// TwinCAT 3 PLC project Untitled1
// ProgramVersion: 3.1.4023.0
// libraries:
//   Tc2_MC2, * (Beckhoff Automation GmbH)
//   Tc2_Standard, * (Beckhoff Automation GmbH)
//   Tc2_System, * (Beckhoff Automation GmbH)
//   Tc3_Module, * (Beckhoff Automation GmbH)
// project tree:
//   DUTs/ AirPiston.TcPOU, ClearLinkEIP.TcPOU (not stored), Homing.TcDUT (not stored), PneumaticInsertion.TcPOU, SuctionPad.TcDUT (not stored)
//   / PlcTask.TcTTO
//   POUs/ MAIN.TcPOU, PistonOnly.TcPOU, WithinTolerance.TcPOU (not stored)
// real-time tasks:
//   TASK PlcTask: cycle T#10ms, priority 20, ADS port 350

CONFIGURATION Untitled1
    RESOURCE PLC ON TwinCAT3
        TASK PlcTask(INTERVAL := T#10ms, PRIORITY := 20);
        PROGRAM MAIN WITH PlcTask : MAIN;
    END_RESOURCE
END_CONFIGURATION

// ---- POUs/MAIN.TcPOU
PROGRAM MAIN
VAR
	insertion : PneumaticInsertion;
	
	enable : BOOL;
	up : BOOL;
	down : BOOL;
	
	in : BOOL;
	out : BOOL;
	
	suction : ARRAY[1..4] OF SuctionPad;
	enableAllSuction : BOOL;
	i : INT;
END_VAR

PistonOnly(smc := insertion.screw);

(*
insertion(
	enable:= enable, 
	slider=> , 
	screw=> , 
	contact=> , 
	home=> , 
	ready=> , 
	busy=> , 
	error=> , 
	homeSet=> );

IF NOT insertion.screw.homeSet THEN
	insertion.homingSequence();
	RETURN;
END_IF

insertion.stop();
	
IF in THEN
	insertion.press();
	out := FALSE;
END_IF

IF out THEN
	insertion.release();
	in := FALSE;
END_IF

IF up THEN
	insertion.slideContinuous(direction:= MC_Positive_Direction);
	down := FALSE;
END_IF

IF down THEN
	insertion.slideContinuous(direction:= MC_Negative_Direction);
	up := FALSE;
END_IF

IF enableAllSuction THEN
	FOR i:=1 TO 4 BY 1 DO
		suction[i].enable := TRUE;
	END_FOR
END_IF
*)

END_PROGRAM

// ---- DUTs/PneumaticInsertion.TcPOU
FUNCTION_BLOCK PneumaticInsertion// EXTENDS Insertion
VAR_INPUT
	enable : BOOL;
END_VAR
VAR_OUTPUT
	slider : ClearLinkEIP;
	screw : AirPiston;
	
	contact : BOOL;
	
	home : BOOL;
	ready : BOOL;
	busy : BOOL;
	error : BOOL;
	
	homeSet : BOOL;
END_VAR

slider(
	bEnable:= enable, 
	home=> , 
	outerLimit=> , 
	innerLimit=> , 
	contact=> contact, 
	homeSet=> );
	
screw(
	bEnable:= enable,
	valveExtend=> , 
	valveRetract=> , 
	contact=> , 
	home=> , 
	innerLimit=> , 
	ready=> , 
	busy=> , 
	error=> , 
	homeSet=> );
	
home := screw.home AND slider.home;
busy := slider.busy OR screw.busy;
error := slider.error OR screw.error;

homeSet := slider.homeSet AND screw.homeSet;

METHOD homingSequence : BOOL
IF NOT screw.homeSet THEN
	screw.homingSequence();
END_IF

homingSequence := slider.homeSet (*AND screw.homeSet*);
END_METHOD

METHOD press : BOOL
VAR_INPUT
	//direction : BOOL; //direction (F = inwards, T = outwards)
	//distance : DINT;
END_VAR
press := screw.extend();
END_METHOD

METHOD release : BOOL
VAR_INPUT
END_VAR
release := screw.retract();
END_METHOD

METHOD slideAbsolute : BOOL
VAR_INPUT
	targetPos : REAL;
END_VAR
slideAbsolute := slider.moveAbsolute(newTarget:= targetPos);
END_METHOD

METHOD slideContinuous : BOOL
VAR_INPUT
	direction : MC_Direction;
END_VAR
slideContinuous := slider.moveContinuous(direction := direction);
END_METHOD

METHOD stop : BOOL
VAR_INPUT
END_VAR
slider.stop();
screw.stop();
END_METHOD

END_FUNCTION_BLOCK

// ---- DUTs/AirPiston.TcPOU
FUNCTION_BLOCK AirPiston
VAR_INPUT CONSTANT
	bEnable : BOOL;
END_VAR
VAR_OUTPUT
	valveExtend AT %Q* : BOOL;
	valveRetract AT %Q* : BOOL;
	
	contact AT %I* : BOOL;
	
	home AT %I* : BOOL;
	innerLimit AT %I* : BOOL;
	
	ready : BOOL;
	busy : BOOL;
	error : BOOL;
	homeSet : BOOL;
END_VAR
VAR
	brakeMode : (PULSE, VARIABLE) := PULSE;
	brakePulse : TP;
	
	step : Homing;
	mode : (HOLD, IN, OUT, REVERSAL);
END_VAR
VAR_STAT CONSTANT
	brakeTime : TIME := T#500MS;
END_VAR

IF NOT bEnable THEN
	stop();
	RETURN;
END_IF

brakePulse(IN:= , PT:= brakeTime, Q=> , ET=> ); //reversal to act as brake
brakePulse.IN := brakePulse.IN AND brakePulse.Q; //automatically turn off pulse

IF home AND valveRetract THEN
	mode := HOLD;
	
ELSIF (innerLimit OR contact) AND valveExtend THEN
	
	IF brakeMode = PULSE THEN
		brakePulse.IN := TRUE; //start reversal to sensor inner limit
		mode := HOLD;
		
	ELSIF brakeMode = VARIABLE THEN
		mode := REVERSAL;
		//RETURN;
		
	END_IF
	
END_IF

CASE mode OF
	HOLD:
		valveExtend := FALSE;
		valveRetract := FALSE;
		
	IN:
		valveExtend := TRUE;
		valveRetract := FALSE;
		
	OUT:
		valveExtend := FALSE;
		valveRetract := TRUE;
		
	REVERSAL:		
		valveExtend := FALSE;
		valveRetract := TRUE;
		
		IF innerLimit THEN
			mode := HOLD;
		END_IF
		
END_CASE

valveRetract := valveRetract OR brakePulse.Q; //from mode or brake

METHOD extend : BOOL
VAR_INPUT
END_VAR
mode := IN;
END_METHOD

METHOD homingSequence : BOOL
(*
this version of homing always traverses to the inner limit before returning to home,
eliminating the possibility of reaching the outer limit while homing
*)
CASE step OF
	Homing.IDLE:
		step := Homing.HOME_OUT;
		
	Homing.REDO: //technically HOME_IN, towards travel limit
		mode := IN;
		
		IF innerLimit THEN
			mode := OUT;
			step := Homing.HOME_OUT;
		END_IF
		
	Homing.HOME_OUT: //towards home
		mode := OUT;
		
		IF home THEN //if reached home
			mode := HOLD;
			step := Homing.DONE;
		END_IF
		
	Homing.DONE:
		mode := HOLD;
		homeSet := TRUE;
		
		homingSequence := TRUE;		
	
END_CASE
END_METHOD

METHOD retract : BOOL
VAR_INPUT
END_VAR
mode := OUT;
END_METHOD

METHOD stop : BOOL
VAR_INPUT
END_VAR
valveExtend := FALSE;
valveRetract := FALSE;
mode := HOLD;
END_METHOD

END_FUNCTION_BLOCK

// ---- POUs/PistonOnly.TcPOU
PROGRAM PistonOnly
VAR_IN_OUT
	smc : AirPiston;
END_VAR
VAR
	ready : BOOL;
	in : BOOL;
	out : BOOL;
END_VAR

smc.bEnable := TRUE;

smc();

IF NOT ready THEN
	ready := smc.homingSequence();
	RETURN;
END_IF


//IF NOT (in OR out) THEN
	//smc.stop();
//END_IF

IF in THEN
	smc.extend();
	out := FALSE;
END_IF

IF out THEN
	smc.retract();
	in := FALSE;
END_IF

IF smc.innerLimit THEN
	in := FALSE;
END_IF

IF smc.home THEN
	out := FALSE;
END_IF

END_PROGRAM
